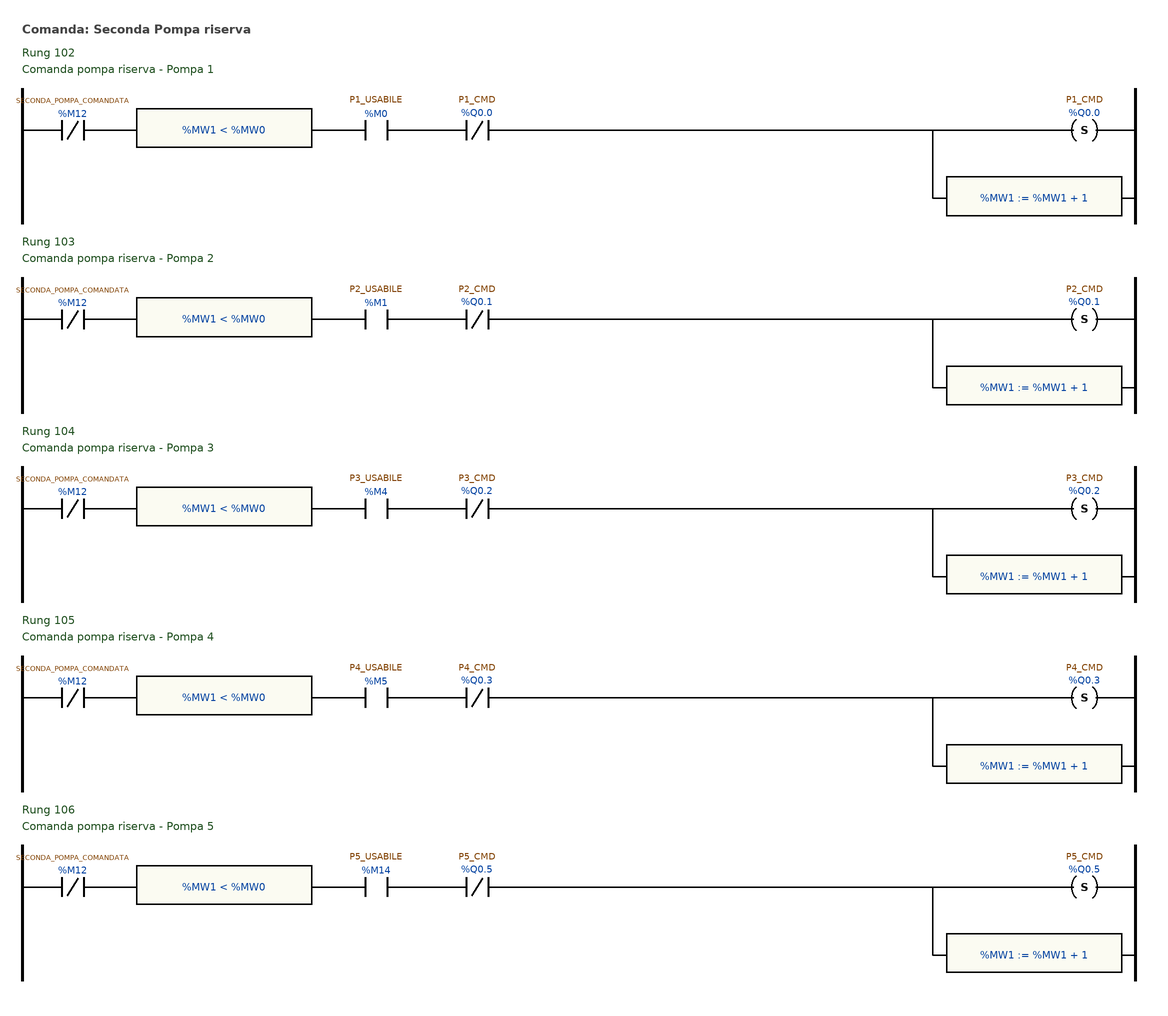
[picture p24: Comanda: Seconda Pompa riserva, ladder]

// Rung 102
// Comanda pompa riserva - Pompa 1
  LDN %M12                (* SECONDA_POMPA_COMANDATA *)
  AND [ %MW1 < %MW0 ]     (* NUM_POMPE_COMANDATE, NUM_POMPE_DA_COMANDARE *)
  AND %M0                 (* P1_USABILE *)
  ANDN %Q0.0              (* P1_CMD *)
  S %Q0.0                 (* P1_CMD *)
  [ %MW1 := %MW1 + 1 ]    (* NUM_POMPE_COMANDATE, NUM_POMPE_COMANDATE *)
  // as ST:
  //   _t1 := NOT SECONDA_POMPA_COMANDATA AND NUM_POMPE_COMANDATE < NUM_POMPE_DA_COMANDARE AND P1_USABILE AND NOT P1_CMD;
  //   IF _t1 THEN P1_CMD := TRUE; END_IF;
  //   IF _t1 THEN NUM_POMPE_COMANDATE := NUM_POMPE_COMANDATE + 1; END_IF;

// Rung 103
// Comanda pompa riserva - Pompa 2
  LDN %M12                (* SECONDA_POMPA_COMANDATA *)
  AND [ %MW1 < %MW0 ]     (* NUM_POMPE_COMANDATE, NUM_POMPE_DA_COMANDARE *)
  AND %M1                 (* P2_USABILE *)
  ANDN %Q0.1              (* P2_CMD *)
  S %Q0.1                 (* P2_CMD *)
  [ %MW1 := %MW1 + 1 ]    (* NUM_POMPE_COMANDATE, NUM_POMPE_COMANDATE *)
  // as ST:
  //   _t1 := NOT SECONDA_POMPA_COMANDATA AND NUM_POMPE_COMANDATE < NUM_POMPE_DA_COMANDARE AND P2_USABILE AND NOT P2_CMD;
  //   IF _t1 THEN P2_CMD := TRUE; END_IF;
  //   IF _t1 THEN NUM_POMPE_COMANDATE := NUM_POMPE_COMANDATE + 1; END_IF;

// Rung 104
// Comanda pompa riserva - Pompa 3
  LDN %M12                (* SECONDA_POMPA_COMANDATA *)
  AND [ %MW1 < %MW0 ]     (* NUM_POMPE_COMANDATE, NUM_POMPE_DA_COMANDARE *)
  AND %M4                 (* P3_USABILE *)
  ANDN %Q0.2              (* P3_CMD *)
  S %Q0.2                 (* P3_CMD *)
  [ %MW1 := %MW1 + 1 ]    (* NUM_POMPE_COMANDATE, NUM_POMPE_COMANDATE *)
  // as ST:
  //   _t1 := NOT SECONDA_POMPA_COMANDATA AND NUM_POMPE_COMANDATE < NUM_POMPE_DA_COMANDARE AND P3_USABILE AND NOT P3_CMD;
  //   IF _t1 THEN P3_CMD := TRUE; END_IF;
  //   IF _t1 THEN NUM_POMPE_COMANDATE := NUM_POMPE_COMANDATE + 1; END_IF;

// Rung 105
// Comanda pompa riserva - Pompa 4
  LDN %M12                (* SECONDA_POMPA_COMANDATA *)
  AND [ %MW1 < %MW0 ]     (* NUM_POMPE_COMANDATE, NUM_POMPE_DA_COMANDARE *)
  AND %M5                 (* P4_USABILE *)
  ANDN %Q0.3              (* P4_CMD *)
  S %Q0.3                 (* P4_CMD *)
  [ %MW1 := %MW1 + 1 ]    (* NUM_POMPE_COMANDATE, NUM_POMPE_COMANDATE *)
  // as ST:
  //   _t1 := NOT SECONDA_POMPA_COMANDATA AND NUM_POMPE_COMANDATE < NUM_POMPE_DA_COMANDARE AND P4_USABILE AND NOT P4_CMD;
  //   IF _t1 THEN P4_CMD := TRUE; END_IF;
  //   IF _t1 THEN NUM_POMPE_COMANDATE := NUM_POMPE_COMANDATE + 1; END_IF;

// Rung 106
// Comanda pompa riserva - Pompa 5
  LDN %M12                (* SECONDA_POMPA_COMANDATA *)
  AND [ %MW1 < %MW0 ]     (* NUM_POMPE_COMANDATE, NUM_POMPE_DA_COMANDARE *)
  AND %M14                (* P5_USABILE *)
  ANDN %Q0.5              (* P5_CMD *)
  S %Q0.5                 (* P5_CMD *)
  [ %MW1 := %MW1 + 1 ]    (* NUM_POMPE_COMANDATE, NUM_POMPE_COMANDATE *)
  // as ST:
  //   _t1 := NOT SECONDA_POMPA_COMANDATA AND NUM_POMPE_COMANDATE < NUM_POMPE_DA_COMANDARE AND P5_USABILE AND NOT P5_CMD;
  //   IF _t1 THEN P5_CMD := TRUE; END_IF;
  //   IF _t1 THEN NUM_POMPE_COMANDATE := NUM_POMPE_COMANDATE + 1; END_IF;

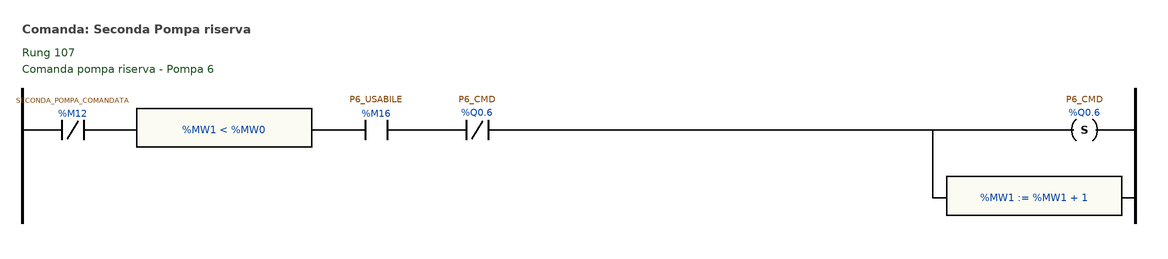

// Rung 107
// Comanda pompa riserva - Pompa 6
  LDN %M12                (* SECONDA_POMPA_COMANDATA *)
  AND [ %MW1 < %MW0 ]     (* NUM_POMPE_COMANDATE, NUM_POMPE_DA_COMANDARE *)
  AND %M16                (* P6_USABILE *)
  ANDN %Q0.6              (* P6_CMD *)
  S %Q0.6                 (* P6_CMD *)
  [ %MW1 := %MW1 + 1 ]    (* NUM_POMPE_COMANDATE, NUM_POMPE_COMANDATE *)
  // as ST:
  //   _t1 := NOT SECONDA_POMPA_COMANDATA AND NUM_POMPE_COMANDATE < NUM_POMPE_DA_COMANDARE AND P6_USABILE AND NOT P6_CMD;
  //   IF _t1 THEN P6_CMD := TRUE; END_IF;
  //   IF _t1 THEN NUM_POMPE_COMANDATE := NUM_POMPE_COMANDATE + 1; END_IF;

Subroutine Comanda: Terza Pompa riserva
  (* SectionNumber=14, Number=12 *)

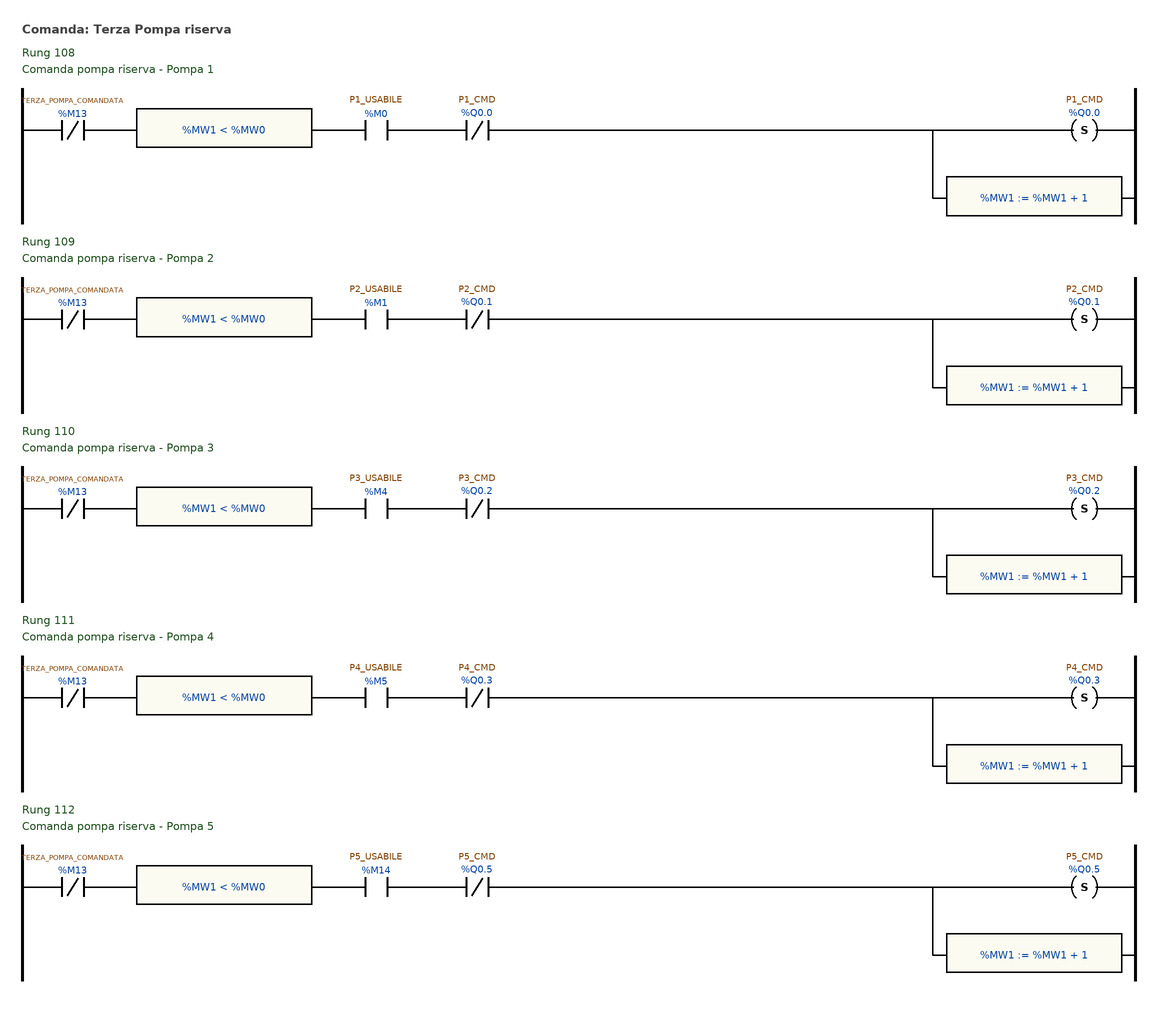

// Rung 108
// Comanda pompa riserva - Pompa 1
  LDN %M13                (* TERZA_POMPA_COMANDATA *)
  AND [ %MW1 < %MW0 ]     (* NUM_POMPE_COMANDATE, NUM_POMPE_DA_COMANDARE *)
  AND %M0                 (* P1_USABILE *)
  ANDN %Q0.0              (* P1_CMD *)
  S %Q0.0                 (* P1_CMD *)
  [ %MW1 := %MW1 + 1 ]    (* NUM_POMPE_COMANDATE, NUM_POMPE_COMANDATE *)
  // as ST:
  //   _t1 := NOT TERZA_POMPA_COMANDATA AND NUM_POMPE_COMANDATE < NUM_POMPE_DA_COMANDARE AND P1_USABILE AND NOT P1_CMD;
  //   IF _t1 THEN P1_CMD := TRUE; END_IF;
  //   IF _t1 THEN NUM_POMPE_COMANDATE := NUM_POMPE_COMANDATE + 1; END_IF;

// Rung 109
// Comanda pompa riserva - Pompa 2
  LDN %M13                (* TERZA_POMPA_COMANDATA *)
  AND [ %MW1 < %MW0 ]     (* NUM_POMPE_COMANDATE, NUM_POMPE_DA_COMANDARE *)
  AND %M1                 (* P2_USABILE *)
  ANDN %Q0.1              (* P2_CMD *)
  S %Q0.1                 (* P2_CMD *)
  [ %MW1 := %MW1 + 1 ]    (* NUM_POMPE_COMANDATE, NUM_POMPE_COMANDATE *)
  // as ST:
  //   _t1 := NOT TERZA_POMPA_COMANDATA AND NUM_POMPE_COMANDATE < NUM_POMPE_DA_COMANDARE AND P2_USABILE AND NOT P2_CMD;
  //   IF _t1 THEN P2_CMD := TRUE; END_IF;
  //   IF _t1 THEN NUM_POMPE_COMANDATE := NUM_POMPE_COMANDATE + 1; END_IF;

// Rung 110
// Comanda pompa riserva - Pompa 3
  LDN %M13                (* TERZA_POMPA_COMANDATA *)
  AND [ %MW1 < %MW0 ]     (* NUM_POMPE_COMANDATE, NUM_POMPE_DA_COMANDARE *)
  AND %M4                 (* P3_USABILE *)
  ANDN %Q0.2              (* P3_CMD *)
  S %Q0.2                 (* P3_CMD *)
  [ %MW1 := %MW1 + 1 ]    (* NUM_POMPE_COMANDATE, NUM_POMPE_COMANDATE *)
  // as ST:
  //   _t1 := NOT TERZA_POMPA_COMANDATA AND NUM_POMPE_COMANDATE < NUM_POMPE_DA_COMANDARE AND P3_USABILE AND NOT P3_CMD;
  //   IF _t1 THEN P3_CMD := TRUE; END_IF;
  //   IF _t1 THEN NUM_POMPE_COMANDATE := NUM_POMPE_COMANDATE + 1; END_IF;

// Rung 111
// Comanda pompa riserva - Pompa 4
  LDN %M13                (* TERZA_POMPA_COMANDATA *)
  AND [ %MW1 < %MW0 ]     (* NUM_POMPE_COMANDATE, NUM_POMPE_DA_COMANDARE *)
  AND %M5                 (* P4_USABILE *)
  ANDN %Q0.3              (* P4_CMD *)
  S %Q0.3                 (* P4_CMD *)
  [ %MW1 := %MW1 + 1 ]    (* NUM_POMPE_COMANDATE, NUM_POMPE_COMANDATE *)
  // as ST:
  //   _t1 := NOT TERZA_POMPA_COMANDATA AND NUM_POMPE_COMANDATE < NUM_POMPE_DA_COMANDARE AND P4_USABILE AND NOT P4_CMD;
  //   IF _t1 THEN P4_CMD := TRUE; END_IF;
  //   IF _t1 THEN NUM_POMPE_COMANDATE := NUM_POMPE_COMANDATE + 1; END_IF;

// Rung 112
// Comanda pompa riserva - Pompa 5
  LDN %M13                (* TERZA_POMPA_COMANDATA *)
  AND [ %MW1 < %MW0 ]     (* NUM_POMPE_COMANDATE, NUM_POMPE_DA_COMANDARE *)
  AND %M14                (* P5_USABILE *)
  ANDN %Q0.5              (* P5_CMD *)
  S %Q0.5                 (* P5_CMD *)
  [ %MW1 := %MW1 + 1 ]    (* NUM_POMPE_COMANDATE, NUM_POMPE_COMANDATE *)
  // as ST:
  //   _t1 := NOT TERZA_POMPA_COMANDATA AND NUM_POMPE_COMANDATE < NUM_POMPE_DA_COMANDARE AND P5_USABILE AND NOT P5_CMD;
  //   IF _t1 THEN P5_CMD := TRUE; END_IF;
  //   IF _t1 THEN NUM_POMPE_COMANDATE := NUM_POMPE_COMANDATE + 1; END_IF;

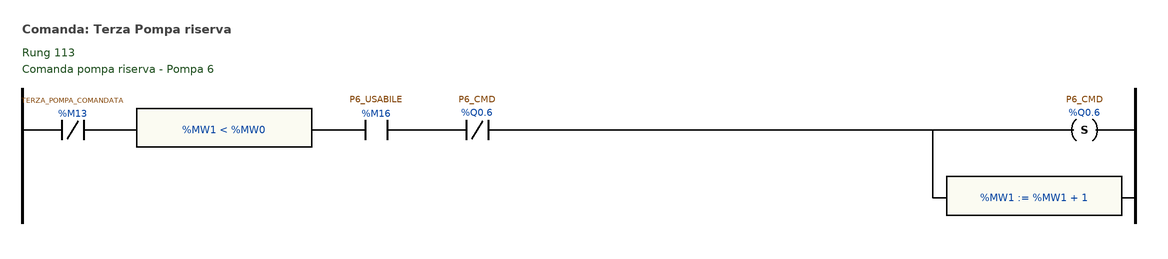

// Rung 113
// Comanda pompa riserva - Pompa 6
  LDN %M13                (* TERZA_POMPA_COMANDATA *)
  AND [ %MW1 < %MW0 ]     (* NUM_POMPE_COMANDATE, NUM_POMPE_DA_COMANDARE *)
  AND %M16                (* P6_USABILE *)
  ANDN %Q0.6              (* P6_CMD *)
  S %Q0.6                 (* P6_CMD *)
  [ %MW1 := %MW1 + 1 ]    (* NUM_POMPE_COMANDATE, NUM_POMPE_COMANDATE *)
  // as ST:
  //   _t1 := NOT TERZA_POMPA_COMANDATA AND NUM_POMPE_COMANDATE < NUM_POMPE_DA_COMANDARE AND P6_USABILE AND NOT P6_CMD;
  //   IF _t1 THEN P6_CMD := TRUE; END_IF;
  //   IF _t1 THEN NUM_POMPE_COMANDATE := NUM_POMPE_COMANDATE + 1; END_IF;

Subroutine Aggiorna Strategia
  (* SectionNumber=15, Number=13 *)

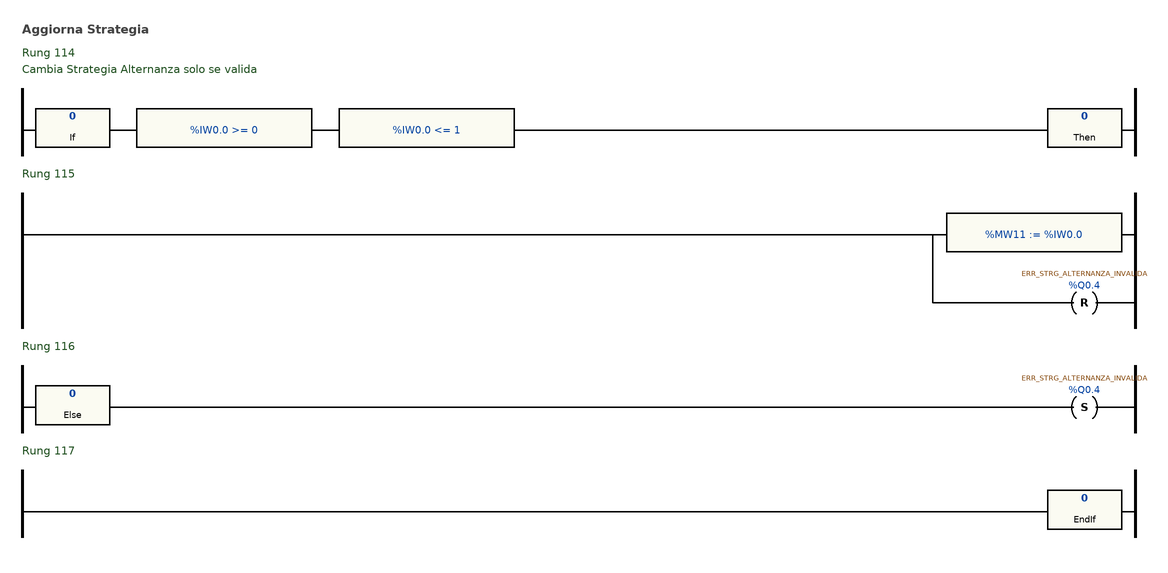

// Rung 114
// Cambia Strategia Alternanza solo se valida
  IF0
  AND [ %IW0.0 >= 0 ]     (* STRG_ALTERNANZA_INPUT *)
  AND [ %IW0.0 <= 1 ]     (* STRG_ALTERNANZA_INPUT *)
  THEN0

// Rung 115
  LD 1
  [ %MW11 := %IW0.0 ]     (* STRG_ALTERNANZA_ATTUALE, STRG_ALTERNANZA_INPUT *)
  R %Q0.4                 (* ERR_STRG_ALTERNANZA_INVALIDA *)
  // as ST:
  //   STRG_ALTERNANZA_ATTUALE := STRG_ALTERNANZA_INPUT;
  //   ERR_STRG_ALTERNANZA_INVALIDA := FALSE;

// Rung 116
  ELSE0
  S %Q0.4                 (* ERR_STRG_ALTERNANZA_INVALIDA *)

// Rung 117
  LD 1
  ENDIF0

Subroutine Ordine: Quarta Pompa
  (* SectionNumber=16, Number=14 *)

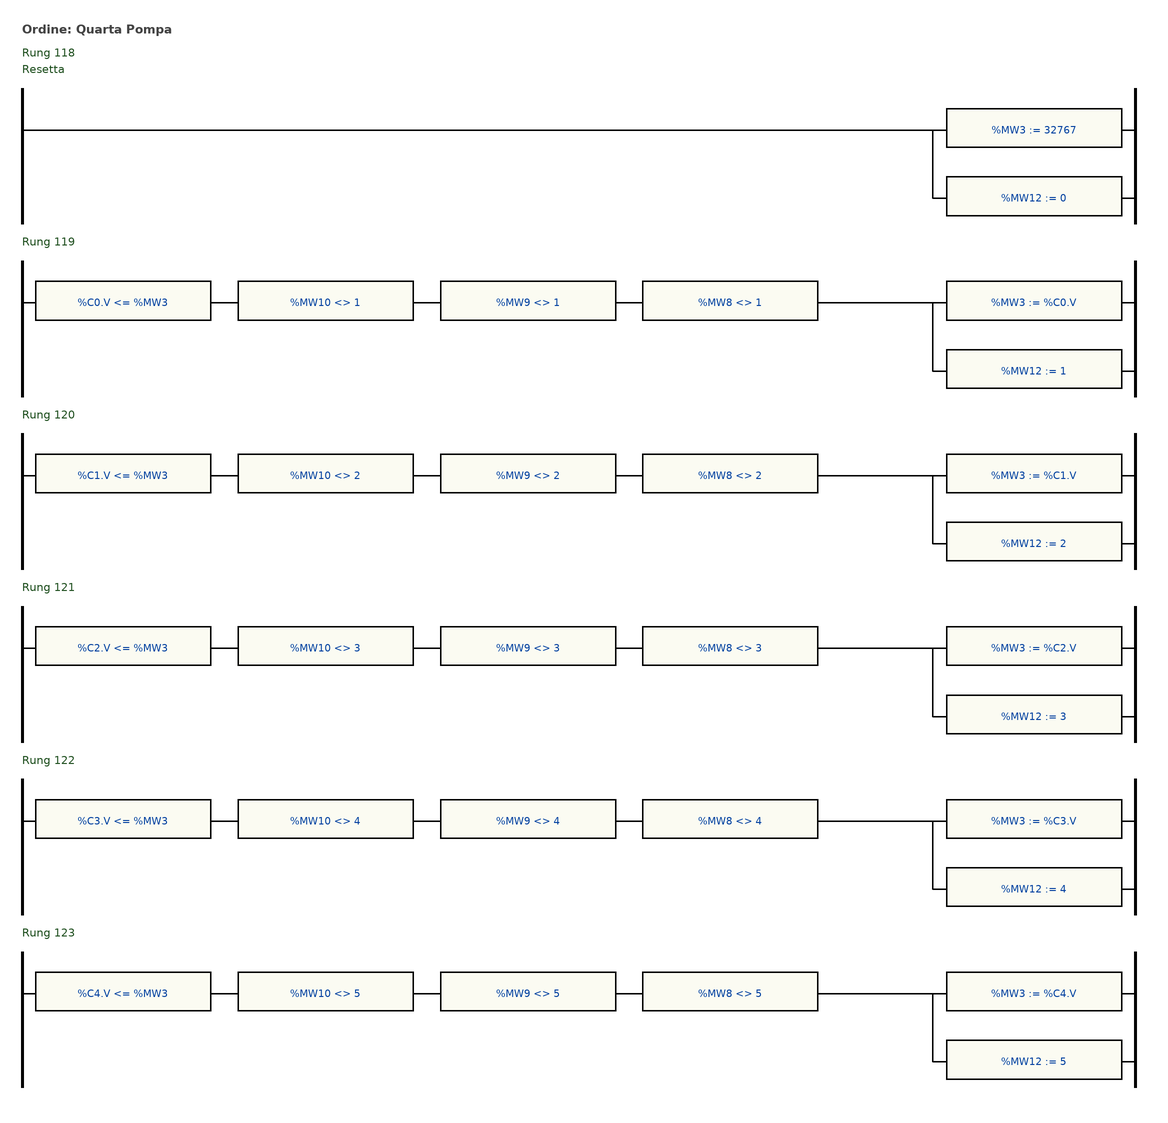

// Rung 118
// Resetta
  LD 1
  [ %MW3 := 32767 ]       (* ULTIMO_MINOR_SECONDI_LAVORATI *)
  [ %MW12 := 0 ]          (* ORDINE_QUARTA_POMPA *)
  // as ST:
  //   ULTIMO_MINOR_SECONDI_LAVORATI := 32767;
  //   ORDINE_QUARTA_POMPA := 0;

// Rung 119
  LD [ %C0.V <= %MW3 ]    (* CONTATORE_P1_SECONDI_LAVORATI, ULTIMO_MINOR_SECONDI_LAVORATI *)
  AND [ %MW10 <> 1 ]      (* ORDINE_TERZA_POMPA *)
  AND [ %MW9 <> 1 ]       (* ORDINE_SECONDA_POMPA *)
  AND [ %MW8 <> 1 ]       (* ORDINE_PRIMA_POMPA *)
  [ %MW3 := %C0.V ]       (* ULTIMO_MINOR_SECONDI_LAVORATI, CONTATORE_P1_SECONDI_LAVORATI *)
  [ %MW12 := 1 ]          (* ORDINE_QUARTA_POMPA *)
  // as ST:
  //   _t1 := CONTATORE_P1_SECONDI_LAVORATI.V <= ULTIMO_MINOR_SECONDI_LAVORATI AND ORDINE_TERZA_POMPA <> 1 AND ORDINE_SECONDA_POMPA <> 1 AND ORDINE_PRIMA_POMPA <> 1;
  //   IF _t1 THEN ULTIMO_MINOR_SECONDI_LAVORATI := CONTATORE_P1_SECONDI_LAVORATI.V; END_IF;
  //   IF _t1 THEN ORDINE_QUARTA_POMPA := 1; END_IF;

// Rung 120
  LD [ %C1.V <= %MW3 ]    (* CONTATORE_P2_SECONDI_LAVORATI, ULTIMO_MINOR_SECONDI_LAVORATI *)
  AND [ %MW10 <> 2 ]      (* ORDINE_TERZA_POMPA *)
  AND [ %MW9 <> 2 ]       (* ORDINE_SECONDA_POMPA *)
  AND [ %MW8 <> 2 ]       (* ORDINE_PRIMA_POMPA *)
  [ %MW3 := %C1.V ]       (* ULTIMO_MINOR_SECONDI_LAVORATI, CONTATORE_P2_SECONDI_LAVORATI *)
  [ %MW12 := 2 ]          (* ORDINE_QUARTA_POMPA *)
  // as ST:
  //   _t1 := CONTATORE_P2_SECONDI_LAVORATI.V <= ULTIMO_MINOR_SECONDI_LAVORATI AND ORDINE_TERZA_POMPA <> 2 AND ORDINE_SECONDA_POMPA <> 2 AND ORDINE_PRIMA_POMPA <> 2;
  //   IF _t1 THEN ULTIMO_MINOR_SECONDI_LAVORATI := CONTATORE_P2_SECONDI_LAVORATI.V; END_IF;
  //   IF _t1 THEN ORDINE_QUARTA_POMPA := 2; END_IF;

// Rung 121
  LD [ %C2.V <= %MW3 ]    (* CONTATORE_P3_SECONDI_LAVORATI, ULTIMO_MINOR_SECONDI_LAVORATI *)
  AND [ %MW10 <> 3 ]      (* ORDINE_TERZA_POMPA *)
  AND [ %MW9 <> 3 ]       (* ORDINE_SECONDA_POMPA *)
  AND [ %MW8 <> 3 ]       (* ORDINE_PRIMA_POMPA *)
  [ %MW3 := %C2.V ]       (* ULTIMO_MINOR_SECONDI_LAVORATI, CONTATORE_P3_SECONDI_LAVORATI *)
  [ %MW12 := 3 ]          (* ORDINE_QUARTA_POMPA *)
  // as ST:
  //   _t1 := CONTATORE_P3_SECONDI_LAVORATI.V <= ULTIMO_MINOR_SECONDI_LAVORATI AND ORDINE_TERZA_POMPA <> 3 AND ORDINE_SECONDA_POMPA <> 3 AND ORDINE_PRIMA_POMPA <> 3;
  //   IF _t1 THEN ULTIMO_MINOR_SECONDI_LAVORATI := CONTATORE_P3_SECONDI_LAVORATI.V; END_IF;
  //   IF _t1 THEN ORDINE_QUARTA_POMPA := 3; END_IF;

// Rung 122
  LD [ %C3.V <= %MW3 ]    (* CONTATORE_P4_SECONDI_LAVORATI, ULTIMO_MINOR_SECONDI_LAVORATI *)
  AND [ %MW10 <> 4 ]      (* ORDINE_TERZA_POMPA *)
  AND [ %MW9 <> 4 ]       (* ORDINE_SECONDA_POMPA *)
  AND [ %MW8 <> 4 ]       (* ORDINE_PRIMA_POMPA *)
  [ %MW3 := %C3.V ]       (* ULTIMO_MINOR_SECONDI_LAVORATI, CONTATORE_P4_SECONDI_LAVORATI *)
  [ %MW12 := 4 ]          (* ORDINE_QUARTA_POMPA *)
  // as ST:
  //   _t1 := CONTATORE_P4_SECONDI_LAVORATI.V <= ULTIMO_MINOR_SECONDI_LAVORATI AND ORDINE_TERZA_POMPA <> 4 AND ORDINE_SECONDA_POMPA <> 4 AND ORDINE_PRIMA_POMPA <> 4;
  //   IF _t1 THEN ULTIMO_MINOR_SECONDI_LAVORATI := CONTATORE_P4_SECONDI_LAVORATI.V; END_IF;
  //   IF _t1 THEN ORDINE_QUARTA_POMPA := 4; END_IF;

// Rung 123
  LD [ %C4.V <= %MW3 ]    (* CONTATORE_P5_SECONDI_LAVORATI, ULTIMO_MINOR_SECONDI_LAVORATI *)
  AND [ %MW10 <> 5 ]      (* ORDINE_TERZA_POMPA *)
  AND [ %MW9 <> 5 ]       (* ORDINE_SECONDA_POMPA *)
  AND [ %MW8 <> 5 ]       (* ORDINE_PRIMA_POMPA *)
  [ %MW3 := %C4.V ]       (* ULTIMO_MINOR_SECONDI_LAVORATI, CONTATORE_P5_SECONDI_LAVORATI *)
  [ %MW12 := 5 ]          (* ORDINE_QUARTA_POMPA *)
  // as ST:
  //   _t1 := CONTATORE_P5_SECONDI_LAVORATI.V <= ULTIMO_MINOR_SECONDI_LAVORATI AND ORDINE_TERZA_POMPA <> 5 AND ORDINE_SECONDA_POMPA <> 5 AND ORDINE_PRIMA_POMPA <> 5;
  //   IF _t1 THEN ULTIMO_MINOR_SECONDI_LAVORATI := CONTATORE_P5_SECONDI_LAVORATI.V; END_IF;
  //   IF _t1 THEN ORDINE_QUARTA_POMPA := 5; END_IF;

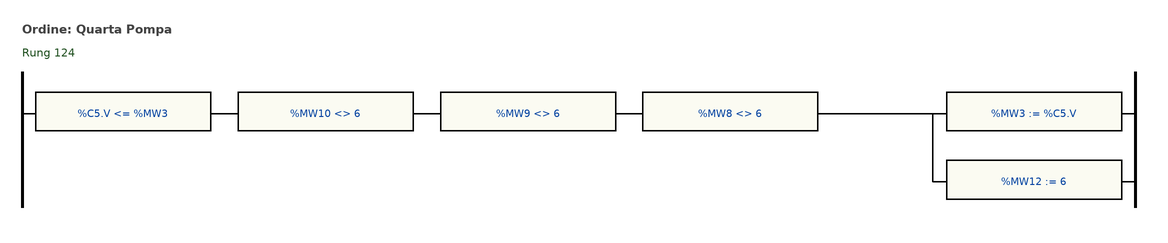

// Rung 124
  LD [ %C5.V <= %MW3 ]    (* CONTATORE_P6_SECONDI_LAVORATI, ULTIMO_MINOR_SECONDI_LAVORATI *)
  AND [ %MW10 <> 6 ]      (* ORDINE_TERZA_POMPA *)
  AND [ %MW9 <> 6 ]       (* ORDINE_SECONDA_POMPA *)
  AND [ %MW8 <> 6 ]       (* ORDINE_PRIMA_POMPA *)
  [ %MW3 := %C5.V ]       (* ULTIMO_MINOR_SECONDI_LAVORATI, CONTATORE_P6_SECONDI_LAVORATI *)
  [ %MW12 := 6 ]          (* ORDINE_QUARTA_POMPA *)
  // as ST:
  //   _t1 := CONTATORE_P6_SECONDI_LAVORATI.V <= ULTIMO_MINOR_SECONDI_LAVORATI AND ORDINE_TERZA_POMPA <> 6 AND ORDINE_SECONDA_POMPA <> 6 AND ORDINE_PRIMA_POMPA <> 6;
  //   IF _t1 THEN ULTIMO_MINOR_SECONDI_LAVORATI := CONTATORE_P6_SECONDI_LAVORATI.V; END_IF;
  //   IF _t1 THEN ORDINE_QUARTA_POMPA := 6; END_IF;

Subroutine Comanda: Quarta Pompa
  (* SectionNumber=17, Number=15 *)

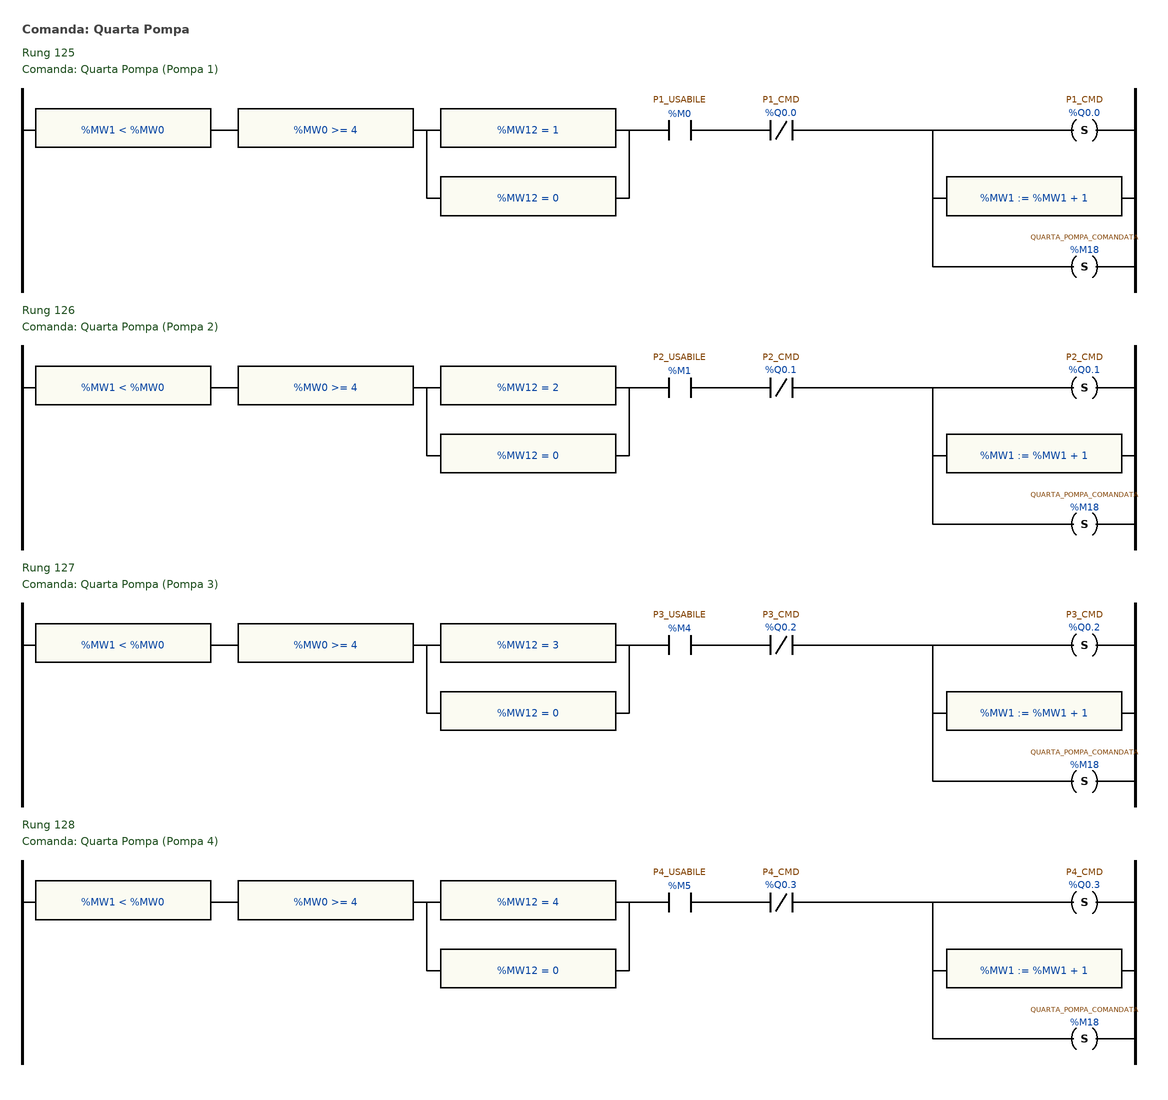

// Rung 125
// Comanda: Quarta Pompa (Pompa 1)
  LD [ %MW1 < %MW0 ]      (* NUM_POMPE_COMANDATE, NUM_POMPE_DA_COMANDARE *)
  AND [ %MW0 >= 4 ]       (* NUM_POMPE_DA_COMANDARE *)
  AND( [ %MW12 = 1 ]      (* ORDINE_QUARTA_POMPA *)
  OR [ %MW12 = 0 ]        (* ORDINE_QUARTA_POMPA *)
  )
  AND %M0                 (* P1_USABILE *)
  ANDN %Q0.0              (* P1_CMD *)
  S %Q0.0                 (* P1_CMD *)
  [ %MW1 := %MW1 + 1 ]    (* NUM_POMPE_COMANDATE, NUM_POMPE_COMANDATE *)
  S %M18                  (* QUARTA_POMPA_COMANDATA *)
  // as ST:
  //   _t1 := NUM_POMPE_COMANDATE < NUM_POMPE_DA_COMANDARE AND NUM_POMPE_DA_COMANDARE >= 4 AND (ORDINE_QUARTA_POMPA = 1 OR ORDINE_QUARTA_POMPA = 0) AND P1_USABILE AND NOT P1_CMD;
  //   IF _t1 THEN P1_CMD := TRUE; END_IF;
  //   IF _t1 THEN NUM_POMPE_COMANDATE := NUM_POMPE_COMANDATE + 1; END_IF;
  //   IF _t1 THEN QUARTA_POMPA_COMANDATA := TRUE; END_IF;

// Rung 126
// Comanda: Quarta Pompa (Pompa 2)
  LD [ %MW1 < %MW0 ]      (* NUM_POMPE_COMANDATE, NUM_POMPE_DA_COMANDARE *)
  AND [ %MW0 >= 4 ]       (* NUM_POMPE_DA_COMANDARE *)
  AND( [ %MW12 = 2 ]      (* ORDINE_QUARTA_POMPA *)
  OR [ %MW12 = 0 ]        (* ORDINE_QUARTA_POMPA *)
  )
  AND %M1                 (* P2_USABILE *)
  ANDN %Q0.1              (* P2_CMD *)
  S %Q0.1                 (* P2_CMD *)
  [ %MW1 := %MW1 + 1 ]    (* NUM_POMPE_COMANDATE, NUM_POMPE_COMANDATE *)
  S %M18                  (* QUARTA_POMPA_COMANDATA *)
  // as ST:
  //   _t1 := NUM_POMPE_COMANDATE < NUM_POMPE_DA_COMANDARE AND NUM_POMPE_DA_COMANDARE >= 4 AND (ORDINE_QUARTA_POMPA = 2 OR ORDINE_QUARTA_POMPA = 0) AND P2_USABILE AND NOT P2_CMD;
  //   IF _t1 THEN P2_CMD := TRUE; END_IF;
  //   IF _t1 THEN NUM_POMPE_COMANDATE := NUM_POMPE_COMANDATE + 1; END_IF;
  //   IF _t1 THEN QUARTA_POMPA_COMANDATA := TRUE; END_IF;

// Rung 127
// Comanda: Quarta Pompa (Pompa 3)
  LD [ %MW1 < %MW0 ]      (* NUM_POMPE_COMANDATE, NUM_POMPE_DA_COMANDARE *)
  AND [ %MW0 >= 4 ]       (* NUM_POMPE_DA_COMANDARE *)
  AND( [ %MW12 = 3 ]      (* ORDINE_QUARTA_POMPA *)
  OR [ %MW12 = 0 ]        (* ORDINE_QUARTA_POMPA *)
  )
  AND %M4                 (* P3_USABILE *)
  ANDN %Q0.2              (* P3_CMD *)
  S %Q0.2                 (* P3_CMD *)
  [ %MW1 := %MW1 + 1 ]    (* NUM_POMPE_COMANDATE, NUM_POMPE_COMANDATE *)
  S %M18                  (* QUARTA_POMPA_COMANDATA *)
  // as ST:
  //   _t1 := NUM_POMPE_COMANDATE < NUM_POMPE_DA_COMANDARE AND NUM_POMPE_DA_COMANDARE >= 4 AND (ORDINE_QUARTA_POMPA = 3 OR ORDINE_QUARTA_POMPA = 0) AND P3_USABILE AND NOT P3_CMD;
  //   IF _t1 THEN P3_CMD := TRUE; END_IF;
  //   IF _t1 THEN NUM_POMPE_COMANDATE := NUM_POMPE_COMANDATE + 1; END_IF;
  //   IF _t1 THEN QUARTA_POMPA_COMANDATA := TRUE; END_IF;

// Rung 128
// Comanda: Quarta Pompa (Pompa 4)
  LD [ %MW1 < %MW0 ]      (* NUM_POMPE_COMANDATE, NUM_POMPE_DA_COMANDARE *)
  AND [ %MW0 >= 4 ]       (* NUM_POMPE_DA_COMANDARE *)
  AND( [ %MW12 = 4 ]      (* ORDINE_QUARTA_POMPA *)
  OR [ %MW12 = 0 ]        (* ORDINE_QUARTA_POMPA *)
  )
  AND %M5                 (* P4_USABILE *)
  ANDN %Q0.3              (* P4_CMD *)
  S %Q0.3                 (* P4_CMD *)
  [ %MW1 := %MW1 + 1 ]    (* NUM_POMPE_COMANDATE, NUM_POMPE_COMANDATE *)
  S %M18                  (* QUARTA_POMPA_COMANDATA *)
  // as ST:
  //   _t1 := NUM_POMPE_COMANDATE < NUM_POMPE_DA_COMANDARE AND NUM_POMPE_DA_COMANDARE >= 4 AND (ORDINE_QUARTA_POMPA = 4 OR ORDINE_QUARTA_POMPA = 0) AND P4_USABILE AND NOT P4_CMD;
  //   IF _t1 THEN P4_CMD := TRUE; END_IF;
  //   IF _t1 THEN NUM_POMPE_COMANDATE := NUM_POMPE_COMANDATE + 1; END_IF;
  //   IF _t1 THEN QUARTA_POMPA_COMANDATA := TRUE; END_IF;

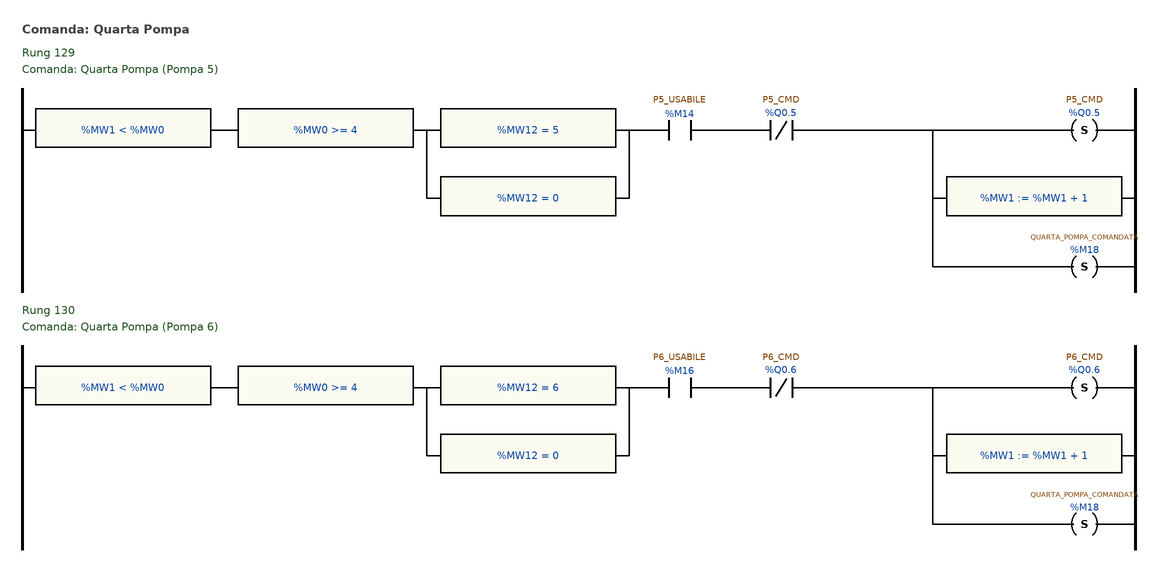

// Rung 129
// Comanda: Quarta Pompa (Pompa 5)
  LD [ %MW1 < %MW0 ]      (* NUM_POMPE_COMANDATE, NUM_POMPE_DA_COMANDARE *)
  AND [ %MW0 >= 4 ]       (* NUM_POMPE_DA_COMANDARE *)
  AND( [ %MW12 = 5 ]      (* ORDINE_QUARTA_POMPA *)
  OR [ %MW12 = 0 ]        (* ORDINE_QUARTA_POMPA *)
  )
  AND %M14                (* P5_USABILE *)
  ANDN %Q0.5              (* P5_CMD *)
  S %Q0.5                 (* P5_CMD *)
  [ %MW1 := %MW1 + 1 ]    (* NUM_POMPE_COMANDATE, NUM_POMPE_COMANDATE *)
  S %M18                  (* QUARTA_POMPA_COMANDATA *)
  // as ST:
  //   _t1 := NUM_POMPE_COMANDATE < NUM_POMPE_DA_COMANDARE AND NUM_POMPE_DA_COMANDARE >= 4 AND (ORDINE_QUARTA_POMPA = 5 OR ORDINE_QUARTA_POMPA = 0) AND P5_USABILE AND NOT P5_CMD;
  //   IF _t1 THEN P5_CMD := TRUE; END_IF;
  //   IF _t1 THEN NUM_POMPE_COMANDATE := NUM_POMPE_COMANDATE + 1; END_IF;
  //   IF _t1 THEN QUARTA_POMPA_COMANDATA := TRUE; END_IF;

// Rung 130
// Comanda: Quarta Pompa (Pompa 6)
  LD [ %MW1 < %MW0 ]      (* NUM_POMPE_COMANDATE, NUM_POMPE_DA_COMANDARE *)
  AND [ %MW0 >= 4 ]       (* NUM_POMPE_DA_COMANDARE *)
  AND( [ %MW12 = 6 ]      (* ORDINE_QUARTA_POMPA *)
  OR [ %MW12 = 0 ]        (* ORDINE_QUARTA_POMPA *)
  )
  AND %M16                (* P6_USABILE *)
  ANDN %Q0.6              (* P6_CMD *)
  S %Q0.6                 (* P6_CMD *)
  [ %MW1 := %MW1 + 1 ]    (* NUM_POMPE_COMANDATE, NUM_POMPE_COMANDATE *)
  S %M18                  (* QUARTA_POMPA_COMANDATA *)
  // as ST:
  //   _t1 := NUM_POMPE_COMANDATE < NUM_POMPE_DA_COMANDARE AND NUM_POMPE_DA_COMANDARE >= 4 AND (ORDINE_QUARTA_POMPA = 6 OR ORDINE_QUARTA_POMPA = 0) AND P6_USABILE AND NOT P6_CMD;
  //   IF _t1 THEN P6_CMD := TRUE; END_IF;
  //   IF _t1 THEN NUM_POMPE_COMANDATE := NUM_POMPE_COMANDATE + 1; END_IF;
  //   IF _t1 THEN QUARTA_POMPA_COMANDATA := TRUE; END_IF;

Subroutine Comanda: Quarta Pompa riserva
  (* SectionNumber=18, Number=16 *)

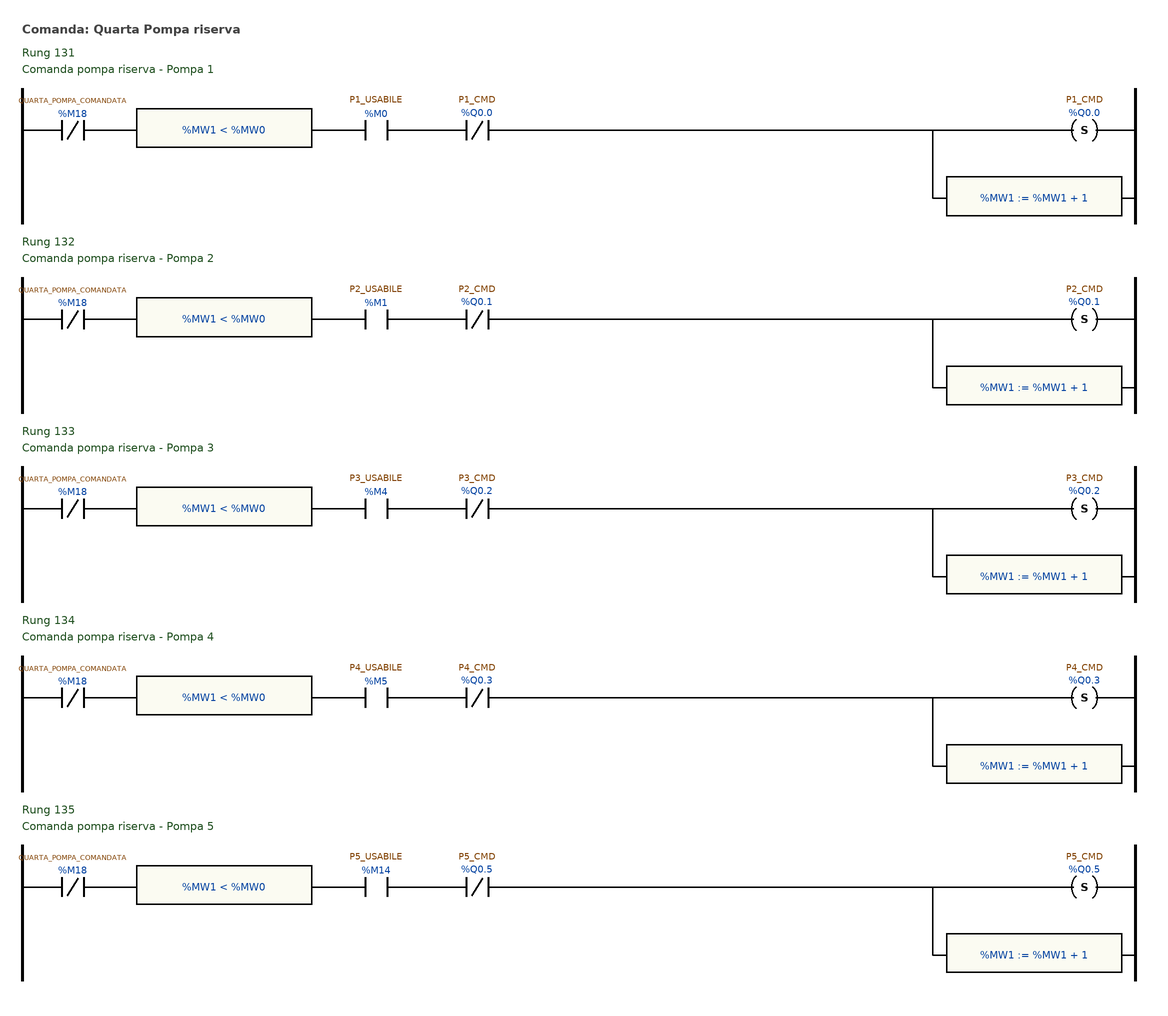

// Rung 131
// Comanda pompa riserva - Pompa 1
  LDN %M18                (* QUARTA_POMPA_COMANDATA *)
  AND [ %MW1 < %MW0 ]     (* NUM_POMPE_COMANDATE, NUM_POMPE_DA_COMANDARE *)
  AND %M0                 (* P1_USABILE *)
  ANDN %Q0.0              (* P1_CMD *)
  S %Q0.0                 (* P1_CMD *)
  [ %MW1 := %MW1 + 1 ]    (* NUM_POMPE_COMANDATE, NUM_POMPE_COMANDATE *)
  // as ST:
  //   _t1 := NOT QUARTA_POMPA_COMANDATA AND NUM_POMPE_COMANDATE < NUM_POMPE_DA_COMANDARE AND P1_USABILE AND NOT P1_CMD;
  //   IF _t1 THEN P1_CMD := TRUE; END_IF;
  //   IF _t1 THEN NUM_POMPE_COMANDATE := NUM_POMPE_COMANDATE + 1; END_IF;

// Rung 132
// Comanda pompa riserva - Pompa 2
  LDN %M18                (* QUARTA_POMPA_COMANDATA *)
  AND [ %MW1 < %MW0 ]     (* NUM_POMPE_COMANDATE, NUM_POMPE_DA_COMANDARE *)
  AND %M1                 (* P2_USABILE *)
  ANDN %Q0.1              (* P2_CMD *)
  S %Q0.1                 (* P2_CMD *)
  [ %MW1 := %MW1 + 1 ]    (* NUM_POMPE_COMANDATE, NUM_POMPE_COMANDATE *)
  // as ST:
  //   _t1 := NOT QUARTA_POMPA_COMANDATA AND NUM_POMPE_COMANDATE < NUM_POMPE_DA_COMANDARE AND P2_USABILE AND NOT P2_CMD;
  //   IF _t1 THEN P2_CMD := TRUE; END_IF;
  //   IF _t1 THEN NUM_POMPE_COMANDATE := NUM_POMPE_COMANDATE + 1; END_IF;

// Rung 133
// Comanda pompa riserva - Pompa 3
  LDN %M18                (* QUARTA_POMPA_COMANDATA *)
  AND [ %MW1 < %MW0 ]     (* NUM_POMPE_COMANDATE, NUM_POMPE_DA_COMANDARE *)
  AND %M4                 (* P3_USABILE *)
  ANDN %Q0.2              (* P3_CMD *)
  S %Q0.2                 (* P3_CMD *)
  [ %MW1 := %MW1 + 1 ]    (* NUM_POMPE_COMANDATE, NUM_POMPE_COMANDATE *)
  // as ST:
  //   _t1 := NOT QUARTA_POMPA_COMANDATA AND NUM_POMPE_COMANDATE < NUM_POMPE_DA_COMANDARE AND P3_USABILE AND NOT P3_CMD;
  //   IF _t1 THEN P3_CMD := TRUE; END_IF;
  //   IF _t1 THEN NUM_POMPE_COMANDATE := NUM_POMPE_COMANDATE + 1; END_IF;

// Rung 134
// Comanda pompa riserva - Pompa 4
  LDN %M18                (* QUARTA_POMPA_COMANDATA *)
  AND [ %MW1 < %MW0 ]     (* NUM_POMPE_COMANDATE, NUM_POMPE_DA_COMANDARE *)
  AND %M5                 (* P4_USABILE *)
  ANDN %Q0.3              (* P4_CMD *)
  S %Q0.3                 (* P4_CMD *)
  [ %MW1 := %MW1 + 1 ]    (* NUM_POMPE_COMANDATE, NUM_POMPE_COMANDATE *)
  // as ST:
  //   _t1 := NOT QUARTA_POMPA_COMANDATA AND NUM_POMPE_COMANDATE < NUM_POMPE_DA_COMANDARE AND P4_USABILE AND NOT P4_CMD;
  //   IF _t1 THEN P4_CMD := TRUE; END_IF;
  //   IF _t1 THEN NUM_POMPE_COMANDATE := NUM_POMPE_COMANDATE + 1; END_IF;

// Rung 135
// Comanda pompa riserva - Pompa 5
  LDN %M18                (* QUARTA_POMPA_COMANDATA *)
  AND [ %MW1 < %MW0 ]     (* NUM_POMPE_COMANDATE, NUM_POMPE_DA_COMANDARE *)
  AND %M14                (* P5_USABILE *)
  ANDN %Q0.5              (* P5_CMD *)
  S %Q0.5                 (* P5_CMD *)
  [ %MW1 := %MW1 + 1 ]    (* NUM_POMPE_COMANDATE, NUM_POMPE_COMANDATE *)
  // as ST:
  //   _t1 := NOT QUARTA_POMPA_COMANDATA AND NUM_POMPE_COMANDATE < NUM_POMPE_DA_COMANDARE AND P5_USABILE AND NOT P5_CMD;
  //   IF _t1 THEN P5_CMD := TRUE; END_IF;
  //   IF _t1 THEN NUM_POMPE_COMANDATE := NUM_POMPE_COMANDATE + 1; END_IF;

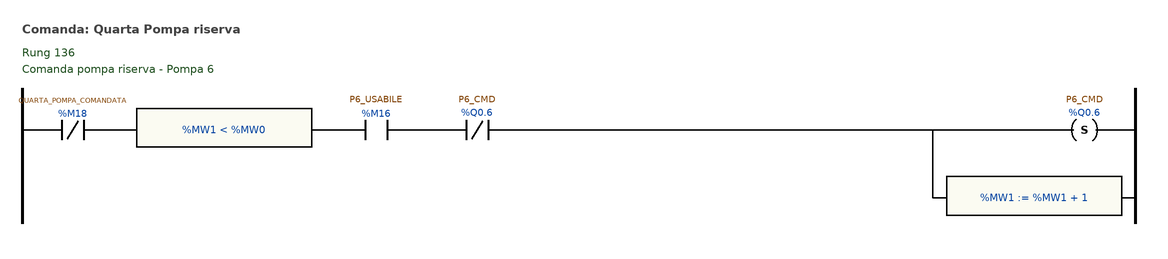

// Rung 136
// Comanda pompa riserva - Pompa 6
  LDN %M18                (* QUARTA_POMPA_COMANDATA *)
  AND [ %MW1 < %MW0 ]     (* NUM_POMPE_COMANDATE, NUM_POMPE_DA_COMANDARE *)
  AND %M16                (* P6_USABILE *)
  ANDN %Q0.6              (* P6_CMD *)
  S %Q0.6                 (* P6_CMD *)
  [ %MW1 := %MW1 + 1 ]    (* NUM_POMPE_COMANDATE, NUM_POMPE_COMANDATE *)
  // as ST:
  //   _t1 := NOT QUARTA_POMPA_COMANDATA AND NUM_POMPE_COMANDATE < NUM_POMPE_DA_COMANDARE AND P6_USABILE AND NOT P6_CMD;
  //   IF _t1 THEN P6_CMD := TRUE; END_IF;
  //   IF _t1 THEN NUM_POMPE_COMANDATE := NUM_POMPE_COMANDATE + 1; END_IF;
